// TwinCAT 3 PLC project PLC01
// ProgramVersion: 3.1.4023.0
// libraries:
//   Tc2_Standard, * (Beckhoff Automation GmbH)
//   Tc2_System, * (Beckhoff Automation GmbH)
//   Tc2_Utilities, * (Beckhoff Automation GmbH)
//   Tc3_Module, * (Beckhoff Automation GmbH)
// project tree:
//   DUTs/ ST_ALARMS.TcDUT, ST_ALARMS_HISTORY.TcDUT, ST_ACTIVE_ALARMS.TcDUT
//   FBs/ FB_DATE_TIME.TcPOU, FB_ALARM_MANAGER.TcPOU
//   / GlobalTextList.TcGTLO, PlcTask.TcTTO, Visualization Manager.TcVMO (not stored), VISU_TASK.TcTTO
//   GVLs/ GVL_ALARMS.TcGVL
//   POUs/ MAIN.TcPOU, PRG_ALARMS.TcPOU
//   VISUs/ ImageList.TcIPO (not stored), MessageList.TcTLO, VISU_ALARMS.TcVIS, VISU_EVENTS.TcVIS, VISU_MAIN.TcVIS
// real-time tasks:
//   TASK PlcTask: cycle T#10ms, priority 20, ADS port 350
//   TASK VISU_TASK: cycle T#200000us, priority 30, ADS port 351

CONFIGURATION PLC01
    RESOURCE PLC ON TwinCAT3
        TASK PlcTask(INTERVAL := T#10ms, PRIORITY := 20);
        TASK VISU_TASK(INTERVAL := T#200000us, PRIORITY := 30);
        PROGRAM MAIN WITH PlcTask : MAIN;
        PROGRAM VisuElems_Visu_Prg WITH VISU_TASK : VisuElems.Visu_Prg;
    END_RESOURCE
END_CONFIGURATION

// ---- DUTs/ST_ALARMS.TcDUT
TYPE ST_ALARMS :
STRUCT
	bActive		: BOOL;		//Alarme ativo
	byGroup		: BYTE;		//Byte que indica o grupo do alarme
	dwTextColor	: DWORD;	//Cor do alarme
END_STRUCT
END_TYPE

// ---- DUTs/ST_ALARMS_HISTORY.TcDUT
TYPE ST_ALARMS_HISTORY:
STRUCT
	byGroup		: BYTE ;		//Byte do grupo
	sDate_on	: STRING(10) ;	//Data de entrada do evento
	sHour_on	: STRING(10) ;	//Hora de entrada do evento
	sDate_off	: STRING(10) ;	//Data de saida do evento
	sHour_off	: STRING(10) ;	//Hora de saida do evento
	iNumber		: INT ;			//Numero da mensagem de alarme
	dwTextColor	: DWORD ;		//Cor do evento
END_STRUCT
END_TYPE

// ---- DUTs/ST_ACTIVE_ALARMS.TcDUT
TYPE ST_ACTIVE_ALARMS :
STRUCT
	byAckStatus	: BYTE;			//Status do alarme
	byGroup		: BYTE;			//Grupo do alarme
	sDate		: STRING(10);	//Hora de entrada do alarme
	sHour		: STRING(10);	//Hora de saida do alarme
	iNumber		: INT;			//Numero do alarme
	dwTextColor	: DWORD;		//Cor do alarme
END_STRUCT
END_TYPE

// ---- GVLs/GVL_ALARMS.TcGVL
VAR_GLOBAL CONSTANT
(* Variaveis constantes do gerenciador de alarmes *)
	
	iNumberOfWarning: INT := 100 ;	//Quantidade de mensagens de alertas 
	iNumberOfAlarms	: INT := 200 ;	//Quantidade de mensagens de alarmes
	iNumberOfEvents	: INT := 300 ;	// = iNumberOfWarning + iNumberOfAlarms;//Total de eventos = alarmes + alertas
	iNumberOfHistory: INT := 1000 ;	//Total de mensagens no historico
END_VAR

VAR_GLOBAL
(* Variaveis para reset de mensagens e array para ativação dos alertas e alarmes *)	
	bResetAlarms		: BOOL ; 										//Reset de Alarmes
	bResetEvents		: BOOL ; 	
	bActiveAlarm		: BOOL ;	//EXISTE ALARME NO SISTEMA / THERE ARE ALARM									//Reset de Eventos
	bActiveWarning		: BOOL ;
	aAlarms				: ARRAY [0..iNumberOfEvents] OF BOOL;				//Cada posição do array ativa uma mensagem de alarme 
END_VAR
	
VAR_GLOBAL PERSISTENT
(* Variaveis do tipo array vinculadas as tabelas de alarme e historico *)	
	ACTIVE_ALARMS	: ARRAY [0..iNumberOfEvents]  OF ST_ACTIVE_ALARMS;		//Array para link com a tabela de alarmes
	HISTORY_ALARMS	: ARRAY [0..iNumberOfHistory] OF ST_ALARMS_HISTORY;		//Array para link com a tabela de eventos
END_VAR

// ---- POUs/MAIN.TcPOU
PROGRAM MAIN
VAR
END_VAR

PRG_ALARMS();	//Chamada do programa Alarmes / call program ALARMS

END_PROGRAM

// ---- POUs/PRG_ALARMS.TcPOU
PROGRAM PRG_ALARMS
VAR
	fbTimer			: TON ; 			//
	fbDateTime		: FB_DATE_TIME;		//
	fbAlarmManager	: FB_ALARM_MANAGER;	//

	_Date : STRING;		//DATA IN STRING FORMAT
	_Time : STRING;		//HOUR IN STRING FORMAT
	
(* Variaveis de exemplo para acionamento dos alarmes *)	
	Condition_01: BOOL;	//TEST TO SIMULATE ALARM 1
	Condition_02: BOOL;	//TEST TO SIMULATE ALARM 2
	Condition_03: BOOL;	//TEST TO SIMULATE EVENT 1
	Condition_04: BOOL;	//TEST TO SIMULATE EVENT 2	
END_VAR

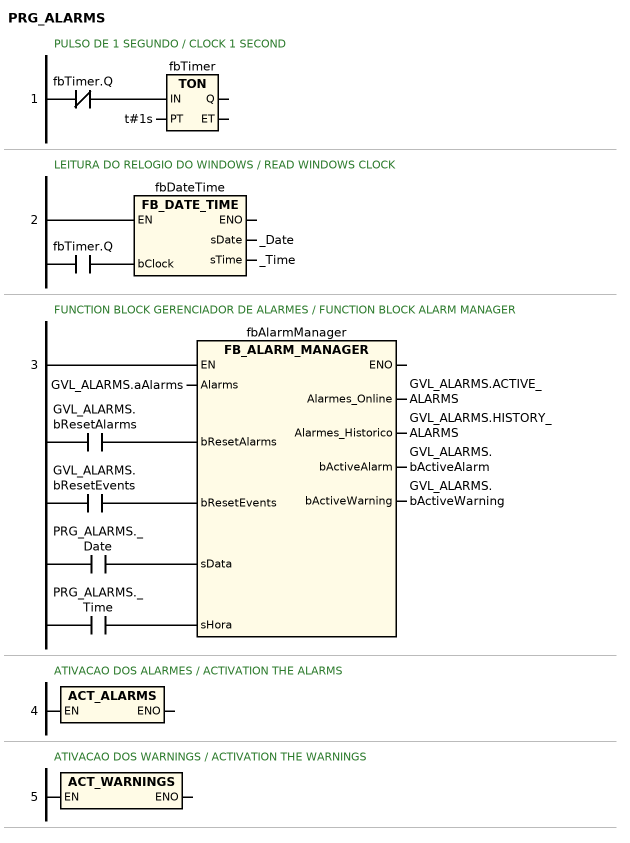
// NETWORK 1
// PULSO DE 1 SEGUNDO / CLOCK 1 SECOND
fbTimer(IN := NOT fbTimer.Q, PT := t#1s); // TON

// NETWORK 2
// LEITURA DO RELOGIO DO WINDOWS / READ WINDOWS CLOCK
fbDateTime(bClock := fbTimer.Q, sDate => _Date, sTime => _Time); // FB_DATE_TIME

// NETWORK 3
// FUNCTION BLOCK GERENCIADOR DE ALARMES / FUNCTION BLOCK ALARM MANAGER
fbAlarmManager(
    Alarms := GVL_ALARMS.aAlarms,
    bResetAlarms := GVL_ALARMS.bResetAlarms,
    bResetEvents := GVL_ALARMS.bResetEvents,
    sData := PRG_ALARMS._Date,
    sHora := PRG_ALARMS._Time,
    Alarmes_Online => GVL_ALARMS.ACTIVE_ALARMS,
    Alarmes_Historico => GVL_ALARMS.HISTORY_ALARMS,
    bActiveAlarm => GVL_ALARMS.bActiveAlarm,
    bActiveWarning => GVL_ALARMS.bActiveWarning); // FB_ALARM_MANAGER

// NETWORK 4
// ATIVACAO DOS ALARMES / ACTIVATION THE ALARMS
ACT_ALARMS();

// NETWORK 5
// ATIVACAO DOS WARNINGS / ACTIVATION THE WARNINGS
ACT_WARNINGS();

ACTION ACT_ALARMS:
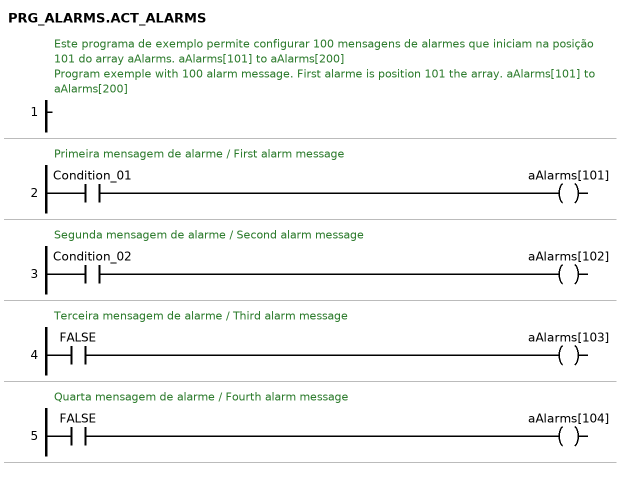
// NETWORK 1
// Este programa de exemplo permite configurar 100 mensagens de alarmes que iniciam na posição 101 do array aAlarms. aAlarms[101] to aAlarms[200]
// Program exemple with 100 alarm message. First alarme is position 101 the array. aAlarms[101] to aAlarms[200]

// NETWORK 2
// Primeira mensagem de alarme / First alarm message
aAlarms[101] := Condition_01;

// NETWORK 3
// Segunda mensagem de alarme / Second alarm message
aAlarms[102] := Condition_02;

// NETWORK 4
// Terceira mensagem de alarme / Third alarm message
aAlarms[103] := FALSE;

// NETWORK 5
// Quarta mensagem de alarme / Fourth alarm message
aAlarms[104] := FALSE;
END_ACTION

ACTION ACT_WARNINGS:
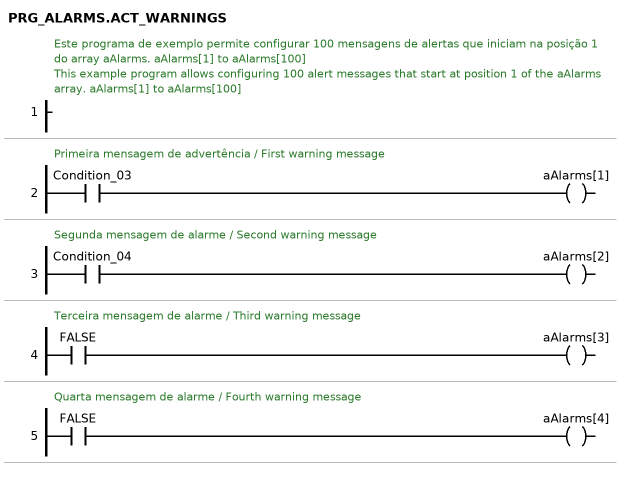
// NETWORK 1
// Este programa de exemplo permite configurar 100 mensagens de alertas que iniciam na posição 1 do array aAlarms. aAlarms[1] to aAlarms[100]
// This example program allows configuring 100 alert messages that start at position 1 of the aAlarms array. aAlarms[1] to aAlarms[100]

// NETWORK 2
// Primeira mensagem de advertência / First warning message
aAlarms[1] := Condition_03;

// NETWORK 3
// Segunda mensagem de alarme / Second warning message
aAlarms[2] := Condition_04;

// NETWORK 4
// Terceira mensagem de alarme / Third warning message
aAlarms[3] := FALSE;

// NETWORK 5
// Quarta mensagem de alarme / Fourth warning message
aAlarms[4] := FALSE;
END_ACTION

END_PROGRAM

// ---- FBs/FB_DATE_TIME.TcPOU
FUNCTION_BLOCK FB_DATE_TIME
VAR_INPUT
	bClock : BOOL ;
END_VAR
VAR_OUTPUT
	sDate		: STRING;
	sTime		: STRING;
END_VAR
VAR
	(* Variaveis para controle de data e hora *)
	Timer1s : TON ; 						//Gerador de pulso de 1s
	fbNtGetTime: NT_GetTime;					//Obtem hora do Windows
	stData_Hora: TIMESTRUCT;			//Estrutura com data e hora

	iAux_Dia	: INT;
	sAux_Dia	: STRING;
	
	iAux_Mes	: INT;
	sAux_Mes	: STRING;
	
	sDia_Mes	: STRING;
	sDia_Mes_Aux: STRING;
	
	iAux_Hora	: INT;
	sAux_Hora	: STRING;
	
	iAux_Min	: INT;
	sAux_Min	: STRING;
	
	iAux_Seg	: INT;
	sAux_Seg	: STRING;
	
	sHora_Aux	: STRING;
	sHora		: STRING;
END_VAR

(********** LEITURA DA DATA E HORA DO PLC ***********)	
(********** READ DATE AND TIME FROM PLC **********)
(* Leitura do relógio da CP / Read Clock from PLC *)	
fbNtGetTime(
	NETID:= '',
	START:=  bClock,
	TMOUT:= ,
	BUSY=> ,
	ERR=> ,
	ERRID=> ,
	TIMESTR=>stData_Hora );

(* DIA DO TIMESTRUCT / DAY FROM TIMESTRUCT *)	
iAux_Dia:= WORD_TO_INT(stData_Hora.wDay);
IF (iAux_Dia) < 10 THEN
	sAux_Dia:= CONCAT('0', INT_TO_STRING(iAux_Dia));
	sAux_Dia:= CONCAT(sAux_Dia, '/');
ELSE
	sAux_Dia:=CONCAT(INT_TO_STRING(iAux_Dia),'/');
END_IF

(* Extrai o mes do TIMESTRUCT *)	
iAux_Mes:= WORD_TO_INT(stData_Hora.wMonth);
IF (iAux_Mes) < 10 THEN
	sAux_Mes:= CONCAT('0', INT_TO_STRING(iAux_Mes));
ELSE
	sAux_Mes:=INT_TO_STRING(iAux_Mes);
END_IF

(* Concatena dia, mês e ano *)
sDia_Mes_Aux := CONCAT(sAux_Dia,sAux_Mes);
sDia_Mes:= CONCAT(sDia_Mes_Aux,'/');
sDate	:= CONCAT(sDia_Mes,WORD_TO_STRING(stData_Hora.wYear));

(* Extrai o hora  do TIMESTRUCT *)	
iAux_Hora:= WORD_TO_INT(stData_Hora.wHour);
IF  (iAux_Hora) < 10 THEN
	sAux_Hora:= CONCAT('0', INT_TO_STRING(iAux_Hora));
	sAux_Hora:= CONCAT(sAux_Hora, ':');
ELSE
	sAux_Hora:=CONCAT(INT_TO_STRING(iAux_Hora),':');
END_IF

(* Extrai o minuto  do TIMESTRUCT *)	
iAux_Min:= WORD_TO_INT(stData_Hora.wMinute);
IF (iAux_Min) < 10 THEN
	sAux_Min:= CONCAT('0', INT_TO_STRING(iAux_Min));
ELSE
	sAux_Min:=INT_TO_STRING(iAux_Min);
END_IF

(* Extrai o segundo do TIMESTRUCT *)	
iAux_Seg:= WORD_TO_INT(stData_Hora.wSecond);
IF (iAux_Seg) < 10 THEN
	sAux_Seg:= CONCAT('0', INT_TO_STRING(iAux_Seg));
ELSE
	sAux_Seg:=INT_TO_STRING(iAux_Seg);
END_IF

(* Concatena hora, minuto e segundo *)
sHora_Aux	:= CONCAT(sAux_Hora,sAux_Min);
sHora	:= CONCAT(sHora_Aux,':');
sTime	:= CONCAT(sHora,sAux_Seg);

END_FUNCTION_BLOCK

// ---- FBs/FB_ALARM_MANAGER.TcPOU
FUNCTION_BLOCK FB_ALARM_MANAGER
VAR_INPUT
	Alarms	: ARRAY [0..iNumberOfEvents] OF BOOL;	//
	bResetAlarms	:	BOOL	;	//
	bResetEvents	:	BOOL	;	//
	sData	:	STRING	;	//Data no formato STRING. Saida do bloco FB_DataHora.
	sHora	:	STRING	;	//Hora no formato STRING Saida do bloco FB_DataHora.
END_VAR
VAR_OUTPUT
	Alarmes_Online : ARRAY[0..iNumberOfEvents] OF ST_ACTIVE_ALARMS;
	Alarmes_Historico : ARRAY[0..iNumberOfHistory] OF ST_ALARMS_HISTORY;
	bActiveAlarm : BOOL ;
	bActiveWarning : BOOL ;
END_VAR
VAR
	Alarmes : ARRAY [0..iNumberOfEvents] OF ST_ALARMS;
	i: INT := 0;
	iArray: INT;
	iAlarmesAtivos: INT := 0;
	iVerificaAlarmes: INT := 0;
	iLinha: INT := 0;
	iAux: INT;
	bAlarmeExistente: BOOL;
	byAlertas: BYTE;
	byAlarmes: BYTE;
	byACK: BYTE;

(* Variaveis para cores das mensagens *)	
	dwColorNull: DWORD;
	dwColorAlerta: DWORD;
	dwColorAlarme: DWORD;
	dwColorAlarmeOff: DWORD;
	dwColorAck: DWORD;

(* Bit para logica no primeiro scan *)	
	FirstScan: BOOL;
	teste: INT;
END_VAR

VAR_IN_OUT
END_VAR

(* Definição dos bytes de cada Grupo de Eventos *)
byAlertas 	:= 1; (* Grupo ALERTAS *)
byAlarmes 	:= 2; (* Grupo ALARMES *)
byACK		:= 5; (* Alarme Reconhecido *)

(* Definição das cores em cada condição *)
dwColorNull		:= 16#FF000000; (* Cor Preta *)
dwColorAlerta 	:= 16#FFFFFF00; (* Cor Amarela *)
dwColorAlarme 	:= 16#FFFF0000; (* Cor Vermelha *)
dwColorAlarmeOff:= 16#FF0000FF; (* Cor Azul *)
dwColorAck 		:= 16#FF00FF00; (* Cor Verde *)

FOR i:= 1 TO iNumberOfEvents DO
	Alarmes[i].bActive := Alarms[i];
	IF i <= iNumberOfWarning THEN
		Alarmes[i].byGroup := byAlertas;
		Alarmes[i].dwTextColor := dwColorAlerta;
	ELSIF (i > iNumberOfWarning) AND (i <= iNumberOfEvents) THEN
		Alarmes[i].byGroup := byAlarmes;	
		Alarmes[i].dwTextColor := dwColorAlarme;
	END_IF
END_FOR

(* Primeiro SCAN, verifica se tem algum alarme no histórico que ficou sem informação ao desligar a máquina *)
IF NOT FirstScan THEN
	FOR iLinha:= 0 TO 1000 BY 1 DO
		IF Alarmes_Historico[iLinha].iNumber <> 0 THEN
			IF Alarmes_Historico[iLinha].sDate_off = '' THEN
				Alarmes_Historico[iLinha].sDate_off		:= 'Power OFF';
				Alarmes_Historico[iLinha].sHour_off		:= 'Power OFF';
			END_IF
		END_IF
	END_FOR
	FirstScan := TRUE;
END_IF

IF TRUE THEN
	WHILE iArray < iNumberOfEvents DO
		(*Verifica se o Alarme esta Ativo , caso positivo popula o array de alarmes Online ( que sera mostrado no Grid )*)
		IF Alarmes[iArray].bActive THEN
			iAux := 0;
			WHILE iAux < iNumberOfEvents AND NOT bAlarmeExistente DO
				IF Alarmes_Online[iAux].iNumber = iArray THEN
					bAlarmeExistente := TRUE;
					bActiveAlarm := TRUE ;
					(* Verifica se o alarme voltou a ativar sem ser reconhecido e troca a cor *)
					IF Alarmes_Online[iAux].dwTextColor = dwColorAlarmeOff THEN 
						Alarmes_Online[iAux].dwTextColor := Alarmes[iArray].dwTextColor;
						Alarmes_Online[iAux].byGroup := byAlarmes;
						
						// Se o Alarme ativou novamente, Armazena novamente no histórico
						FOR iLinha:= 1000 TO 1 BY -1 DO
							ALARMES_HISTORICO[iLinha] := ALARMES_HISTORICO[iLinha-1];
						END_FOR
						Alarmes_Historico[0].dwTextColor	:= Alarmes[iArray].dwTextColor;
						Alarmes_Historico[0].sDate_on		:= sData;
						Alarmes_Historico[0].sHour_on		:= sHora;
						Alarmes_Historico[0].sDate_off		:= '';
						Alarmes_Historico[0].sHour_off		:= '';
						Alarmes_Historico[0].iNumber		:= iArray;
						Alarmes_Historico[0].byGroup		:= Alarmes[iArray].byGroup;

					END_IF
				END_IF
				iAux := iAux + 1;
			END_WHILE

			IF NOT bAlarmeExistente THEN
				// Apresentação de um novo alarme
				FOR iLinha:= iAlarmesAtivos TO 1 BY -1 DO
					Alarmes_Online[iLinha] := Alarmes_Online[iLinha-1];
				END_FOR
				Alarmes_Online[0].dwTextColor	:= Alarmes[iArray].dwTextColor;
				Alarmes_Online[0].sDate			:= sData ;
				Alarmes_Online[0].sHour			:= sHora ;
				Alarmes_Online[0].iNumber		:= iArray ;
				Alarmes_Online[0].byAckStatus	:= 0;
				Alarmes_Online[0].byGroup		:= Alarmes[iArray].byGroup;
				
				// Incrementa contagem de alarmes ativos
				iAlarmesAtivos := iAlarmesAtivos+1;

				// Armazena todos os alarmes em histórico
				FOR iLinha:= 1000 TO 1 BY -1 DO
					Alarmes_Historico[iLinha] := Alarmes_Historico[iLinha-1];
				END_FOR
				Alarmes_Historico[0].dwTextColor	:= Alarmes[iArray].dwTextColor;
				Alarmes_Historico[0].sDate_on		:= sData ;
				Alarmes_Historico[0].sHour_on		:= sHora ;
				Alarmes_Historico[0].sDate_off		:= '';
				Alarmes_Historico[0].sHour_off		:= '';
				Alarmes_Historico[0].iNumber		:= iArray;
				Alarmes_Historico[0].byGroup		:= Alarmes[iArray].byGroup;
			END_IF

		END_IF

		iArray := iArray+1;
		bAlarmeExistente := FALSE;
		bActiveAlarm := FALSE ;

	END_WHILE


	WHILE iVerificaAlarmes < iAlarmesAtivos AND iAlarmesAtivos > 0 DO

		IF bResetAlarms THEN
			Alarmes_Online[iVerificaAlarmes].byAckStatus := byACK; (* Alarme foi Reconhecido mas continua ativo *)
			Alarmes_Online[iVerificaAlarmes].dwTextColor := dwColorAck; (* COR Alarme foi Reconhecido mas continua ativo *)
		END_IF
		
		(*Verifica se o Alarme ainda esta Ativo , caso negativo retira do array de alarmes Online ( que sera mostrado no Grid )*)
		IF NOT Alarmes[ Alarmes_Online[iVerificaAlarmes].iNumber ].bActive THEN
			Alarmes_Online[iVerificaAlarmes].dwTextColor := dwColorAlarmeOff; (* COR Alarme Não está mais ativo *)
	
			(* Se o Alarme não está mais ativo, informa o horário que o alarme foi desligado no histórico *)
			FOR iLinha:= 0 TO 1000 BY 1 DO
				IF Alarmes_Historico[iLinha].iNumber = Alarmes_Online[iVerificaAlarmes].iNumber THEN
					IF Alarmes_Historico[iLinha].sDate_off = '' THEN
						Alarmes_Historico[iLinha].sDate_off		:= sData ;
						Alarmes_Historico[iLinha].sHour_off		:= sHora ;
					END_IF
					EXIT;
				END_IF
			END_FOR
			
			IF Alarmes_Online[iVerificaAlarmes].byAckStatus = byACK THEN
			
				FOR iLinha:= iVerificaAlarmes TO (iNumberOfEvents-1) BY 1 DO
					Alarmes_Online[iLinha] := Alarmes_Online[iLinha+1];
				END_FOR

				Alarmes_Online[iNumberOfEvents].sDate		:= '';
				Alarmes_Online[iNumberOfEvents].sHour		:= '';
				Alarmes_Online[iNumberOfEvents].dwTextColor	:= dwColorNull;
				Alarmes_Online[iNumberOfEvents].iNumber		:= 0;
				Alarmes_Online[iNumberOfEvents].byAckStatus	:= 0;
				Alarmes_Online[iNumberOfEvents].byGroup		:= 0;
				iAlarmesAtivos := iAlarmesAtivos -1 ;
			
			END_IF
		
		END_IF

		iVerificaAlarmes := iVerificaAlarmes + 1 ;

	END_WHILE

	IF iArray >= iNumberOfEvents THEN
		iArray				:=0;(*Index Utilizado para navegar o Array de Alarmes para verificar se os alarmes estao OnLine*)
		iVerificaAlarmes	:=0;
		iLinha				:=0;
	END_IF

END_IF

//RESET EVENTS / RESETA EVENTOS
IF bResetEvents THEN (* Reset de eventos *)
	FOR iLinha:= 0 TO iNumberOfHistory BY 1 DO
		Alarmes_Historico[iLinha].byGroup		:= 0 ;	
		Alarmes_Historico[iLinha].sDate_on		:= ' ' ;
		Alarmes_Historico[iLinha].sHour_on		:= ' ' ;
		Alarmes_Historico[iLinha].sDate_off		:= ' ' ;
		Alarmes_Historico[iLinha].sHour_off		:= ' ' ;
		Alarmes_Historico[iLinha].iNumber		:= 0 ;		
		Alarmes_Historico[iLinha].dwTextColor	:= 16#FF000000 ;
	END_FOR
END_IF

//CHECK ACTIVE ALARM / VERIFICA SE EXISTE ALARME ATIVO
FOR i := 0 TO iNumberOfEvents DO
	// Alarme precisa estar ativo no grupo 2 de alarme e Não reconhecido
	IF (Alarmes_Online[i].byGroup = 2) AND (Alarmes_Online[i].byAckStatus <> 5) THEN
		bActiveAlarm := TRUE;
		EXIT;
	ELSE
		bActiveAlarm := FALSE;
	END_IF
	
	IF (Alarmes_Online[i].byGroup = 1) AND (Alarmes_Online[i].byAckStatus <> 5) THEN
		bActiveWarning := TRUE ;
	ELSE
		bActiveWarning := FALSE ;
	END_IF		
END_FOR

END_FUNCTION_BLOCK

// ---- GlobalTextList.TcGTLO
TEXTLIST GlobalTextList
  662 = ' HOUR IN'
  416 = ' IN'
  588 = '!'
  288 = 'ACTIVE_ALARMS[INDEX].byacess'
  394 = 'ACTIVE_ALARMS[INDEX].byAckStatus'
  4 = 'Alarmes Online'
  958 = 'ALARMS'
  64 = 'BACK'
  996 = 'C'
  47 = 'DATA'
  231 = 'DATA IN'
  841 = 'DATA OFF'
  936 = 'DATE'
  692 = 'DATE IN'
  245 = 'DATE OFF'
  3 = 'Exemplo de Alarmes e Eventos'
  2 = 'Historico Alarmes'
  335 = 'HISTORY'
  49 = 'HORA'
  836 = 'HORA IN'
  508 = 'HORA OFF'
  561 = 'HOUR'
  296 = 'HOUR IN'
  606 = 'HOUR OFF'
  16 = 'Limpa Historico'
  735 = 'MENSAGEM'
  134 = 'MESSAGE'
  928 = 'MESSSAGE'
  17 = 'Reconhece Alarmes'
  33 = 'RESET ALARMES'
  477 = 'RESET ALARMS'
  905 = 'RESET EVENTS'
  623 = 'RESET HISTORY'
  8 = 'Tela de Alarmes'
  15 = 'Tela de Histórico'
  292 = 'TIME'
  1 = 'Voltar'
  903 = 'VOLTAR'
END_TEXTLIST

// ---- VISUs/MessageList.TcTLO
TEXTLIST MessageList
  0 = ' '
  1 = 'MENSAGEM DE ADVERTENCIA 01'
  2 = 'MENSAGEM DE ADVERTENCIA 02'
  3 = 'MENSAGEM DE ADVERTENCIA 03'
  4 = 'MENSAGEM DE ADVERTENCIA 04'
  5 = 'MENSAGEM DE ADVERTENCIA 05'
  6 = 'MENSAGEM DE ADVERTENCIA 06'
  7 = 'MENSAGEM DE ADVERTENCIA 07'
  8 = 'MENSAGEM DE ADVERTENCIA 08'
  9 = 'MENSAGEM DE ADVERTENCIA 09'
  10 = 'MENSAGEM DE ADVERTENCIA 10'
  11 = 'MENSAGEM DE ADVERTENCIA ...'
  12 = 'MENSAGEM DE ADVERTENCIA ...'
  13 = 'MENSAGEM DE ADVERTENCIA ...'
  14 = 'MENSAGEM DE ADVERTENCIA ...'
  15 = 'MENSAGEM DE ADVERTENCIA ...'
  99 = 'MENSAGEM DE ADVERTENCIA 99'
  101 = 'MENSAGEM DE ALARME 01'
  102 = 'MENSAGEM DE ALARME 02'
  103 = 'MENSAGEM DE ALARME 03'
  104 = 'MENSAGEM DE ALARME 04'
  105 = 'MENSAGEM DE ALARME 05'
  106 = 'MENSAGEM DE ALARME 06'
  107 = 'MENSAGEM DE ALARME 07'
  108 = 'MENSAGEM DE ALARME 08'
  109 = 'MENSAGEM DE ALARME 09'
  110 = 'MENSAGEM DE ALARME 10'
  111 = 'MENSAGEM DE ALARME ...'
  299 = 'MENSAGEM DE ALARME 299'
   = ''
END_TEXTLIST

// ---- VISUs/VISU_ALARMS.TcVIS
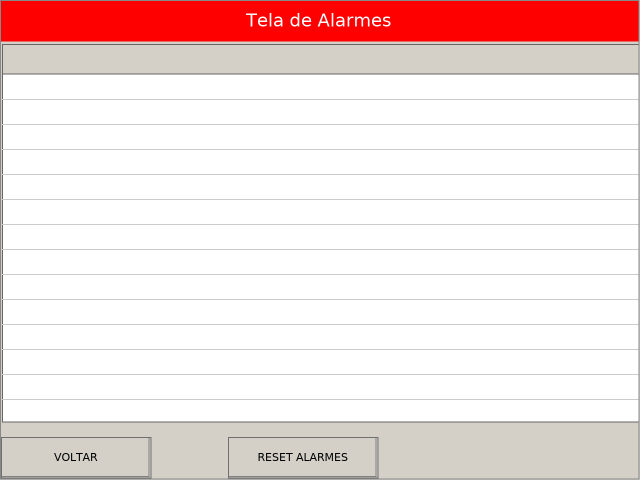
VISUALIZATION VISU_ALARMS  // 640x480
    Button (1,437 150x41), "VOLTAR"
        OnMouseClick: change screen: VISU_MAIN
    Rectangle (-1,0 640x41), "Tela de Alarmes"
    Button (228,437 150x41), "RESET ALARMES"
        tap GVL_ALARMS.bResetAlarms
    Table (2,44 637x378), data array: GVL_ALARMS.ACTIVE_ALARMS
        p746581629: GVL_ALARMS.HISTORY_ALARMS[INDEX].dwTextColor
        p3854506369: GVL_ALARMS.ACTIVE_ALARMS[INDEX].byAckStatus
        p1892666644: GVL_ALARMS.ACTIVE_ALARMS[INDEX].byGroup
        p338671338: ACTIVE_ALARMS[INDEX].sDate
        p2170511999: GVL_ALARMS.ACTIVE_ALARMS[INDEX].sHour
        p3723444502: GVL_ALARMS.ACTIVE_ALARMS[INDEX].iNumber
        p1218418051: GVL_ALARMS.ACTIVE_ALARMS[INDEX].dwTextColor
        p2232123230: !
        p1791247317: GVL_ALARMS.ACTIVE_ALARMS[INDEX].sDate
END_VISUALIZATION

// ---- VISUs/VISU_EVENTS.TcVIS
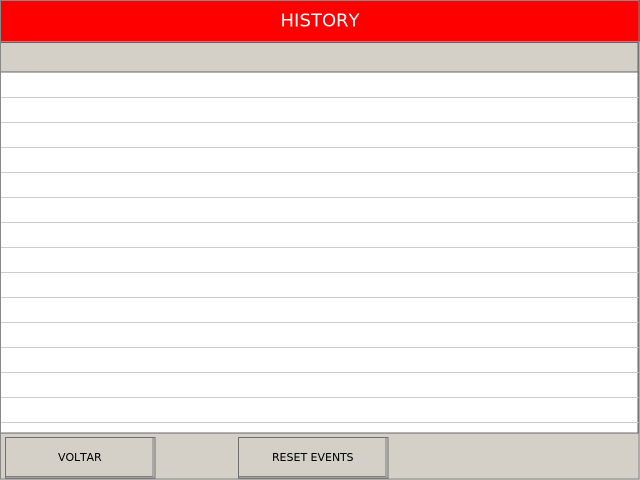
VISUALIZATION VISU_EVENTS  // 640x480
    Button (5,437 150x41), "VOLTAR"
        OnMouseClick: change screen: VISU_MAIN
    Table (0,42 638x391), data array: GVL_ALARMS.HISTORY_ALARMS
        p3854506369: GVL_ALARMS.HISTORY_ALARMS[INDEX].byGroup
        p1892666644: GVL_ALARMS.HISTORY_ALARMS[INDEX].sDate_on
        p338671338: GVL_ALARMS.HISTORY_ALARMS[INDEX].sHour_on
        p2170511999: GVL_ALARMS.HISTORY_ALARMS[INDEX].sDate_off
        p3723444502: GVL_ALARMS.HISTORY_ALARMS[INDEX].sHour_off
        p1218418051: GVL_ALARMS.HISTORY_ALARMS[INDEX].iNumber
        p746581629: GVL_ALARMS.HISTORY_ALARMS[INDEX].dwTextColor
        p511219082: DATA IN
        p1755163831: HORA IN
        p4092479075: DATA OFF
        p2237128397: HORA OFF
    Rectangle (0,0 640x41), "HISTORY"
    Button (238,437 150x41), "RESET EVENTS"
        tap GVL_ALARMS.bResetEvents
END_VISUALIZATION

// ---- VISUs/VISU_MAIN.TcVIS
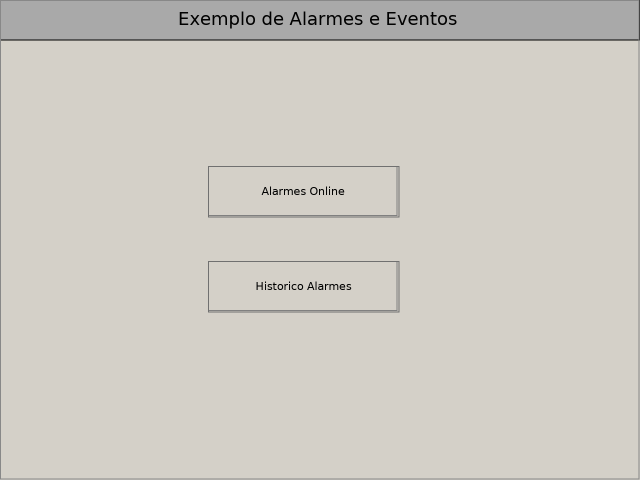
VISUALIZATION VISU_MAIN  // 640x480
    Button (208,261 191x51), "Historico Alarmes"
        OnMouseClick: change screen: VISU_EVENTS
    Rectangle (0,-1 640x41)
    Label (0,4 636x30), "Exemplo de Alarmes e Eventos"
    Button (208,166 191x51), "Alarmes Online"
        OnMouseClick: change screen: VISU_ALARMS
END_VISUALIZATION
